(* PLC project MQTT, Beckhoff Automation GmbH TwinCAT PLC Control 3.5.13.20 *)
(* stored: creationDateTime 2021-01-27T09:58:10.3431314, modificationDateTime 2021-01-27T09:58:10.3431314 *)

PROGRAM PrgMQttSubscribe
VAR_INPUT
	sTopicSub : STRING(255);
END_VAR
VAR
	fbMqttClient : FB_IotMqttClient;
	bSetParameter : BOOL := TRUE;
	bConnect : BOOL := TRUE;
	
	(* received message *)
	bSubscribed : BOOL;
	{attribute 'TcEncoding':='UTF-8'}
	sTopicRcv: STRING(255);
	{attribute 'TcEncoding':='UTF-8'}
	sPayloadRcv : STRING(255);
	fbMessageQueue : FB_IotMqttMessageQueue;
	fbMessage : FB_IotMqttMessage;
	
	hrErrorOccurred : HRESULT; // contains the latest occurred error
END_VAR

            IF bSetParameter THEN
	bSetParameter := FALSE;
	fbMqttClient.sHostName:= GVL_MQTT.mqtt_broker;
	fbMqttClient.nHostPort:= GVL_MQTT.mqtt_port;
	fbMqttClient.sTopicPrefix:= ''; 
	fbMqttClient.sUserName:= GVL_MQTT.username;
	fbMqttClient.sUserPassword:= GVL_MQTT.password;
	
	//Nicht verwendete MQTT Parameter
//	fbMqttClient.nKeepAlive:= 60; 
//	fbMqttClient.sClientId:= 'MyTcMqttClient';  
//	fbMqttClient.stWill:= ; 
//	fbMqttClient.stTLS:= ;
	fbMqttClient.ipMessageQueue := fbMessageQueue;
END_IF

fbMqttClient.Execute(bConnect);
IF fbMqttClient.bError THEN
	// add your error logging here
	hrErrorOccurred := fbMqttClient.hrErrorCode;
END_IF

IF fbMessageQueue.nQueuedMessages > 0 THEN
	IF fbMessageQueue.Dequeue(fbMessage:=fbMessage) THEN
		fbMessage.GetTopic(pTopic:=ADR(sTopicRcv), nTopicSize:=SIZEOF(sTopicRcv) );
		fbMessage.GetPayload(pPayload:=ADR(sPayloadRcv), nPayloadSize:=SIZEOF(sPayloadRcv), bSetNullTermination:=FALSE);
	END_IF
END_IF

IF fbMqttClient.bConnected THEN
	IF NOT bSubscribed THEN
		bSubscribed := fbMqttClient.Subscribe(sTopic:=sTopicSub, eQoS:=TcIotMqttQos.AtMostOnceDelivery);
		IF fbMqttClient.bError THEN
			// add your error logging here
			hrErrorOccurred := fbMqttClient.hrErrorCode;
		END_IF
	END_IF
	
		IF fbMqttClient.bError THEN
			// add your error logging here
			hrErrorOccurred := fbMqttClient.hrErrorCode;
		END_IF
END_IF
          
END_PROGRAM
